SUBAPPLICATION Uebung_094 (* Beispiel für E_PERMIT *)
  (* Standard: 61499-2; Description: Copyright (c) 2023 Meisterschulen am Ostbahnhof This program and the accompanying materials are made available under the terms of the Eclipse Public License 2.0 which is available at https://www.eclipse.org/legal/epl-2.0/ SPDX-License-Identifier: EPL-2.0 Beispiel für E_CTD Aufwärts zählen UAO Curriculum Module 3 - The IEC 61499 Standard, Seite 93 *)
  (* Version 1.0, 2023-10-23, Franz Höpfinger, Meisterschulen am Ostbahnhof *)
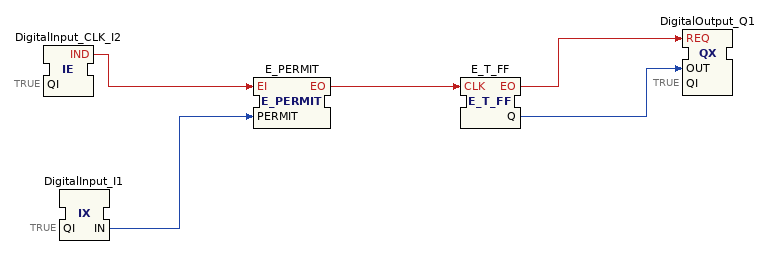
  FBS
    DigitalInput_I1 : IX(QI := TRUE);
    DigitalInput_CLK_I2 : IE(QI := TRUE);
    E_PERMIT : E_PERMIT;
    E_T_FF : E_T_FF;
    DigitalOutput_Q1 : QX(QI := TRUE);
  END_FBS
  EVENT_CONNECTIONS
    DigitalInput_CLK_I2.IND TO E_PERMIT.EI;
    E_T_FF.EO TO DigitalOutput_Q1.REQ;
    E_PERMIT.EO TO E_T_FF.CLK;
  END_CONNECTIONS
  DATA_CONNECTIONS
    DigitalInput_I1.IN TO E_PERMIT.PERMIT;
    E_T_FF.Q TO DigitalOutput_Q1.OUT;
  END_CONNECTIONS
END_SUBAPPLICATION
